FUNCTION_BLOCK AR_MIN (* minimum (OUT = MIN(IN1, IN2)) *)
  (* Standard: 61499-2; Description: Copyright (c) 2026 HR Agrartechnik GmbH This program and the accompanying materials are made available under the terms of the Eclipse Public License 2.0 which is available at https://www.eclipse.org/legal/epl-2.0/ SPDX-License-Identifier: EPL-2.0 *)
  (* Version 1.0, 2026-09-18, Franz Höpfinger, HR Agrartechnik GmbH, initial API and implementation *)
  PACKAGE adapter::iec61131::selection;
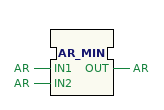
  SOCKETS
    IN1 : adapter::types::unidirectional::AR; (* Input value 1 *)
    IN2 : adapter::types::unidirectional::AR; (* Input value 2 *)
  END_SOCKETS
  PLUGS
    OUT : adapter::types::unidirectional::AR; (* MIN(IN1, IN2) *)
  END_PLUGS
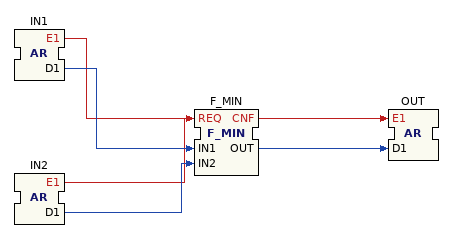
  FBS
    F_MIN : iec61131::selection::F_MIN;
  END_FBS
  EVENT_CONNECTIONS
    F_MIN.CNF TO OUT.E1;
    IN1.E1 TO F_MIN.REQ;
    IN2.E1 TO F_MIN.REQ;
  END_CONNECTIONS
  DATA_CONNECTIONS
    F_MIN.OUT TO OUT.D1;
    IN1.D1 TO F_MIN.IN1;
    IN2.D1 TO F_MIN.IN2;
  END_CONNECTIONS
END_FUNCTION_BLOCK
